// TIA Portal V17 export
// export: Created 2025-03-05T07:59:09.1060697Z, ExportSetting WithDefaults, DisplayName Totally Integrated Automation Portal, DisplayVersion V17 Update 8, DisplayName TIA Portal Openness, DisplayVersion V17 Update 8, DisplayName TIA Portal Version Control Interface, DisplayVersion V17, DisplayName SINAMICS Startdrive Advanced, DisplayVersion V17 SP2, DisplayName SINAMICS Startdrive G110M, G120, G120C, G120D, G120P, G115D, DisplayVersion V17 SP2, DisplayName SINAMICS Startdrive G130, G150, S120, S150, SINAMICS MV, S210, DisplayVersion V17 SP2, DisplayName STEP 7 Professional, DisplayVersion V17 Update 8, DisplayName SINUMERIK ONE STEP 7 Toolbox, DisplayVersion V17 Update 12, DisplayName SINUMERIK 840D sl STEP 7 Toolbox, DisplayVersion V17 Update 12, DisplayName STEP 7 Safety, DisplayVersion V17 Update 6, DisplayName WinCC Advanced, DisplayVersion V17 Update 8
DATA_BLOCK "DB3000_PART_PRESENT_CONTROL_U01_STA_1"   // DB3000
{ S7_Optimized_Access := 'FALSE'; DB_Accessible_From_OPC_UA := 'FALSE' }
VERSION : 0.1
// stored: AutoNumber false, DBAccessibleFromOPCUA false, DBAccessibleFromWebserver true, IsOnlyStoredInLoadMemory false, IsWriteProtectedInAS false
   VAR RETAIN
      NO_PART : Bool;   // UNIT 01 STATION 1 NO PART PRESENT
      FACE_N_PART_PRESENT : Bool;   // UNIT 01 STATION 1 FACE N PART PRESENT
      FACE_R_PART_PRESENT : Bool;   // UNIT 01 STATION 1 FACE R PART PRESENT
      FACE_N_MASTER_PRESENT : Bool := FALSE;   // UNIT 01 STATION 1 FACE N MASTER PRESENT
      FACE_R_MASTER_PRESENT : Bool := FALSE;   // UNIT 01 STATION 1 FACE R MASTER PRESENT
      PART_PRESENT_INPUT : Bool;   // PART PRESENT INPUT
      PART_HAT_POSITION_INPUT : Bool;   // PART HAT POSITION INPUT
      SPARE_BOOL : Array[1..18] of Bool;
   END_VAR
BEGIN
END_DATA_BLOCK
